// TIA Portal V20 export
// export: Created 2026-04-18T06:33:56.704783Z, ExportSetting WithDefaults, DisplayName Totally Integrated Automation Portal, DisplayVersion V20, DisplayName TIA Portal Openness, DisplayVersion V20, DisplayName TIA Portal Version Control Interface, DisplayVersion V20, DisplayName STEP 7 Professional, DisplayVersion V20, DisplayName STEP 7 Safety, DisplayVersion V20, DisplayName WinCC Basic/Comfort/Advanced, DisplayVersion V20
TYPE "UDT_ProcessUnit"
// stored: IsFailsafeCompliant false
   STRUCT
      unitId : Int := 0;
      unitName : String[32] := 'Unit';
      recipeId : Int := 0;
      modules { S7_SetPoint := 'True'} : Array[1..3] of "UDT_EquipmentModule";
   END_STRUCT;
END_TYPE
